// SIMATIC S7-200 project (STEP 7-Micro/WIN), CPU 224 REL 02.01

SYMBOL_TABLE USER1
oneLevel         VW2
twoLevel         VW3
onePres4ma       VW4
onePres20ma      VW5
twoPres4ma       VW6
twoPres20ma      VW7
oneUpp           VW8
oneLww           VW9
twoUpp           VW10
twoLww           VW11
pmp1mode         VW12     // 0 - stop, 1 - auto, 3 - man
pmp2mode         VW13
dOneLevel        VD14
dTwoLevel        VD16
dOnePres4ma      VD18
dOnePres20ma     VD20
dTwoPres4ma      VD22
dTwoPres20ma     VD24
dOneUpp          VD26
dOneLww          VD28
dTwoUpp          VD30
dTwoLww          VD32
pmp1auto         I0.0
pmp2auto         I0.1
pmp1man          I0.2
pmp2man          I0.3
pmp1turn         Q0.0
pmp2turn         Q0.1
oneMustStart     V34.0
twoMustStart     V34.1
pmp1state        V34.2
pmp2state        V34.3
END_SYMBOL_TABLE

ORGANIZATION_BLOCK MAIN:OB1
TITLE=PROGRAM COMMENTS
BEGIN
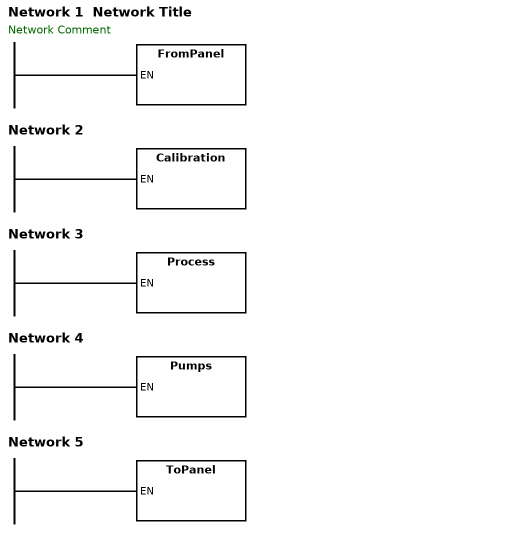
Network 1 // Network Title
// Network Comment
// (network saved uncompiled; LAD cells follow)
// row 0: c0 --  c1 [FromPanel EN:=power@row0]
Network 2
// (network saved uncompiled; LAD cells follow)
// row 0: c0 --  c1 [Calibration EN:=power@row0]
Network 3
// (network saved uncompiled; LAD cells follow)
// row 0: c0 --  c1 [Process EN:=power@row0]
Network 4
// (network saved uncompiled; LAD cells follow)
// row 0: c0 --  c1 [Pumps EN:=power@row0]
Network 5
// (network saved uncompiled; LAD cells follow)
// row 0: c0 --  c1 [ToPanel EN:=power@row0]
END_ORGANIZATION_BLOCK

SUBROUTINE_BLOCK Calibration:SBR0
TITLE=SUBROUTINE COMMENTS
BEGIN
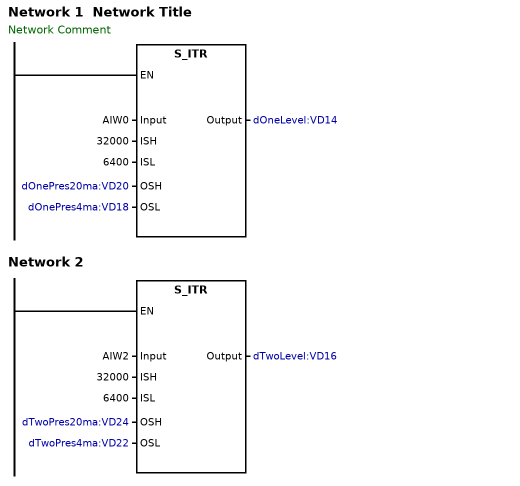
Network 1 // Network Title
// Network Comment
// (network saved uncompiled; LAD cells follow)
// row 0: c0 --  c1 [S_ITR EN:=power@row0, Input:=AIW0, ISH:=32000, ISL:=6400, OSH:=dOnePres20ma:VD20, OSL:=dOnePres4ma:VD18, Output=>dOneLevel:VD14]
// row 1: c1 [box]
// row 2: c1 [box]
Network 2
// (network saved uncompiled; LAD cells follow)
// row 0: c0 --  c1 [S_ITR EN:=power@row0, Input:=AIW2, ISH:=32000, ISL:=6400, OSH:=dTwoPres20ma:VD24, OSL:=dTwoPres4ma:VD22, Output=>dTwoLevel:VD16]
// row 1: c1 [box]
// row 2: c1 [box]
END_SUBROUTINE_BLOCK

SUBROUTINE_BLOCK FromPanel:SBR1
TITLE=SUBROUTINE COMMENTS
BEGIN
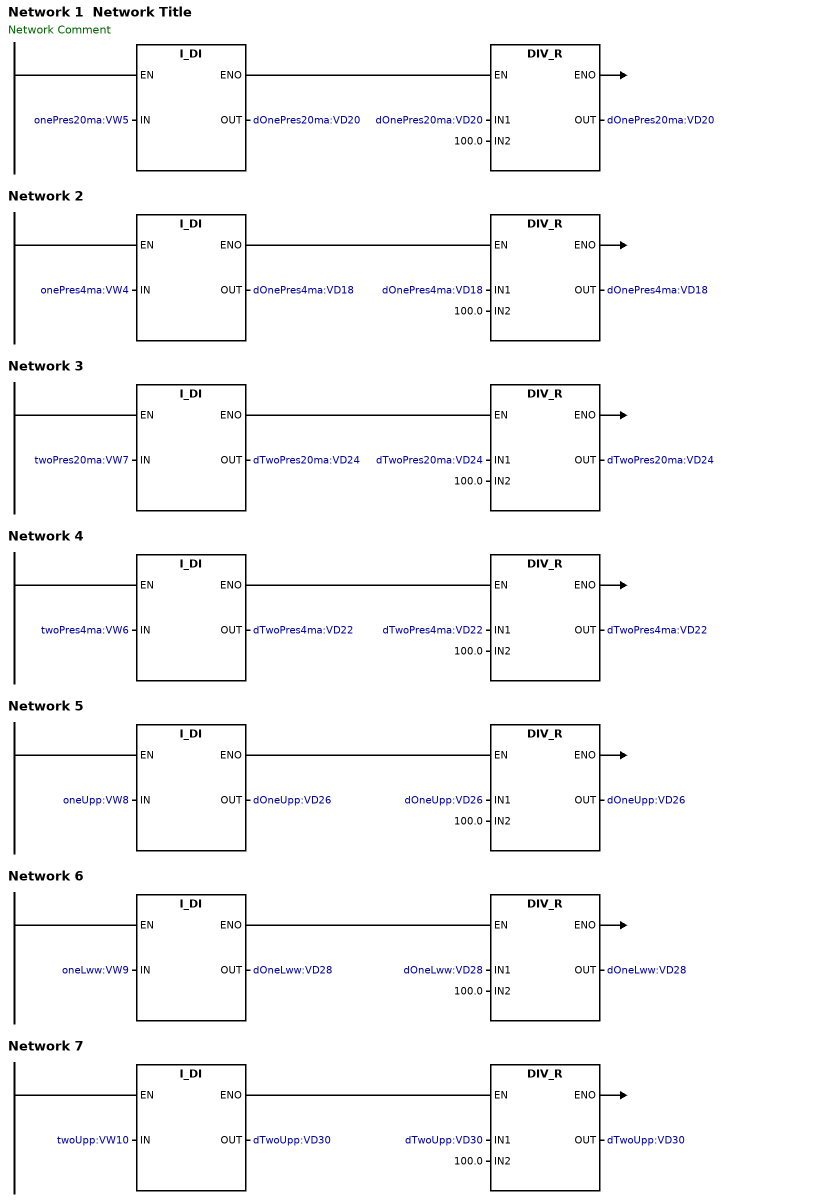
Network 1 // Network Title
// Network Comment
// (network saved uncompiled; LAD cells follow)
// row 0: c0 --  c1 [I_DI EN:=power@row0, IN:=onePres20ma:VW5, ENO=>power, OUT=>dOnePres20ma:VD20]  c2 --  c3 --  c4 [DIV_R EN:=power@row0, IN1:=dOnePres20ma:VD20, IN2:=100.0, ENO=>power, OUT=>dOnePres20ma:VD20]  c5 ->
// row 1: c1 [box]  c4 [box]
Network 2
// (network saved uncompiled; LAD cells follow)
// row 0: c0 --  c1 [I_DI EN:=power@row0, IN:=onePres4ma:VW4, ENO=>power, OUT=>dOnePres4ma:VD18]  c2 --  c3 --  c4 [DIV_R EN:=power@row0, IN1:=dOnePres4ma:VD18, IN2:=100.0, ENO=>power, OUT=>dOnePres4ma:VD18]  c5 ->
// row 1: c1 [box]  c4 [box]
Network 3
// (network saved uncompiled; LAD cells follow)
// row 0: c0 --  c1 [I_DI EN:=power@row0, IN:=twoPres20ma:VW7, ENO=>power, OUT=>dTwoPres20ma:VD24]  c2 --  c3 --  c4 [DIV_R EN:=power@row0, IN1:=dTwoPres20ma:VD24, IN2:=100.0, ENO=>power, OUT=>dTwoPres20ma:VD24]  c5 ->
// row 1: c1 [box]  c4 [box]
Network 4
// (network saved uncompiled; LAD cells follow)
// row 0: c0 --  c1 [I_DI EN:=power@row0, IN:=twoPres4ma:VW6, ENO=>power, OUT=>dTwoPres4ma:VD22]  c2 --  c3 --  c4 [DIV_R EN:=power@row0, IN1:=dTwoPres4ma:VD22, IN2:=100.0, ENO=>power, OUT=>dTwoPres4ma:VD22]  c5 ->
// row 1: c1 [box]  c4 [box]
Network 5
// (network saved uncompiled; LAD cells follow)
// row 0: c0 --  c1 [I_DI EN:=power@row0, IN:=oneUpp:VW8, ENO=>power, OUT=>dOneUpp:VD26]  c2 --  c3 --  c4 [DIV_R EN:=power@row0, IN1:=dOneUpp:VD26, IN2:=100.0, ENO=>power, OUT=>dOneUpp:VD26]  c5 ->
// row 1: c1 [box]  c4 [box]
Network 6
// (network saved uncompiled; LAD cells follow)
// row 0: c0 --  c1 [I_DI EN:=power@row0, IN:=oneLww:VW9, ENO=>power, OUT=>dOneLww:VD28]  c2 --  c3 --  c4 [DIV_R EN:=power@row0, IN1:=dOneLww:VD28, IN2:=100.0, ENO=>power, OUT=>dOneLww:VD28]  c5 ->
// row 1: c1 [box]  c4 [box]
Network 7
// (network saved uncompiled; LAD cells follow)
// row 0: c0 --  c1 [I_DI EN:=power@row0, IN:=twoUpp:VW10, ENO=>power, OUT=>dTwoUpp:VD30]  c2 --  c3 --  c4 [DIV_R EN:=power@row0, IN1:=dTwoUpp:VD30, IN2:=100.0, ENO=>power, OUT=>dTwoUpp:VD30]  c5 ->
// row 1: c1 [box]  c4 [box]
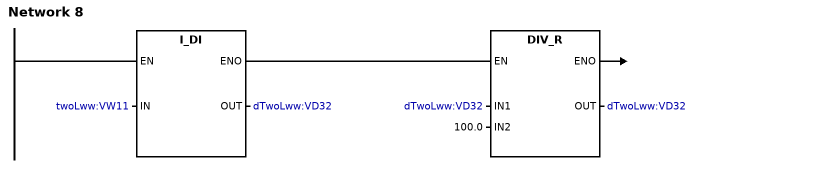
Network 8
// (network saved uncompiled; LAD cells follow)
// row 0: c0 --  c1 [I_DI EN:=power@row0, IN:=twoLww:VW11, ENO=>power, OUT=>dTwoLww:VD32]  c2 --  c3 --  c4 [DIV_R EN:=power@row0, IN1:=dTwoLww:VD32, IN2:=100.0, ENO=>power, OUT=>dTwoLww:VD32]  c5 ->
// row 1: c1 [box]  c4 [box]
END_SUBROUTINE_BLOCK

// SBR2: protected block, not included

SUBROUTINE_BLOCK Process:SBR3
TITLE=SUBROUTINE COMMENTS
BEGIN
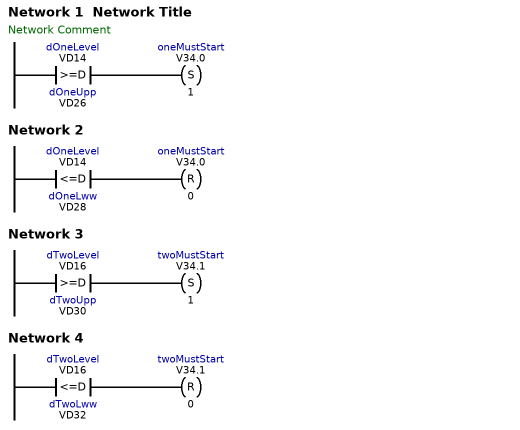
Network 1 // Network Title
// Network Comment
// (network saved uncompiled; LAD cells follow)
// row 0: c0 -|>=D|- dOneLevel:VD14, dOneUpp:VD26  c1 -(S) oneMustStart:V34.0, 1
Network 2
// (network saved uncompiled; LAD cells follow)
// row 0: c0 -|<=D|- dOneLevel:VD14, dOneLww:VD28  c1 -(R) oneMustStart:V34.0, 0
Network 3
// (network saved uncompiled; LAD cells follow)
// row 0: c0 -|>=D|- dTwoLevel:VD16, dTwoUpp:VD30  c1 -(S) twoMustStart:V34.1, 1
Network 4
// (network saved uncompiled; LAD cells follow)
// row 0: c0 -|<=D|- dTwoLevel:VD16, dTwoLww:VD32  c1 -(R) twoMustStart:V34.1, 0
END_SUBROUTINE_BLOCK

SUBROUTINE_BLOCK Pumps:SBR4
TITLE=SUBROUTINE COMMENTS
BEGIN
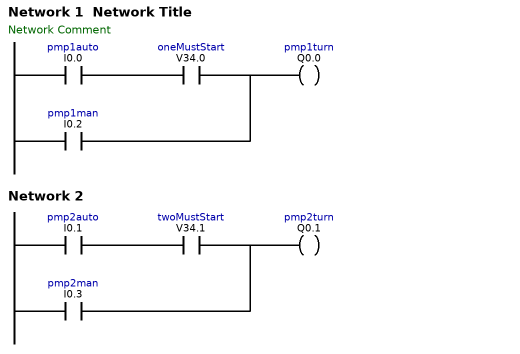
Network 1 // Network Title
// Network Comment
// (network saved uncompiled; LAD cells follow)
// row 0: c0 -| |- pmp1auto:I0.0  c1 -| |- oneMustStart:V34.0 v  c2 -( ) pmp1turn:Q0.0
// row 1: c0 -| |- pmp1man:I0.2  c1 -- ^
Network 2
// (network saved uncompiled; LAD cells follow)
// row 0: c0 -| |- pmp2auto:I0.1  c1 -| |- twoMustStart:V34.1 v  c2 -( ) pmp2turn:Q0.1
// row 1: c0 -| |- pmp2man:I0.3  c1 -- ^
END_SUBROUTINE_BLOCK

SUBROUTINE_BLOCK ToPanel:SBR5
TITLE=SUBROUTINE COMMENTS
BEGIN
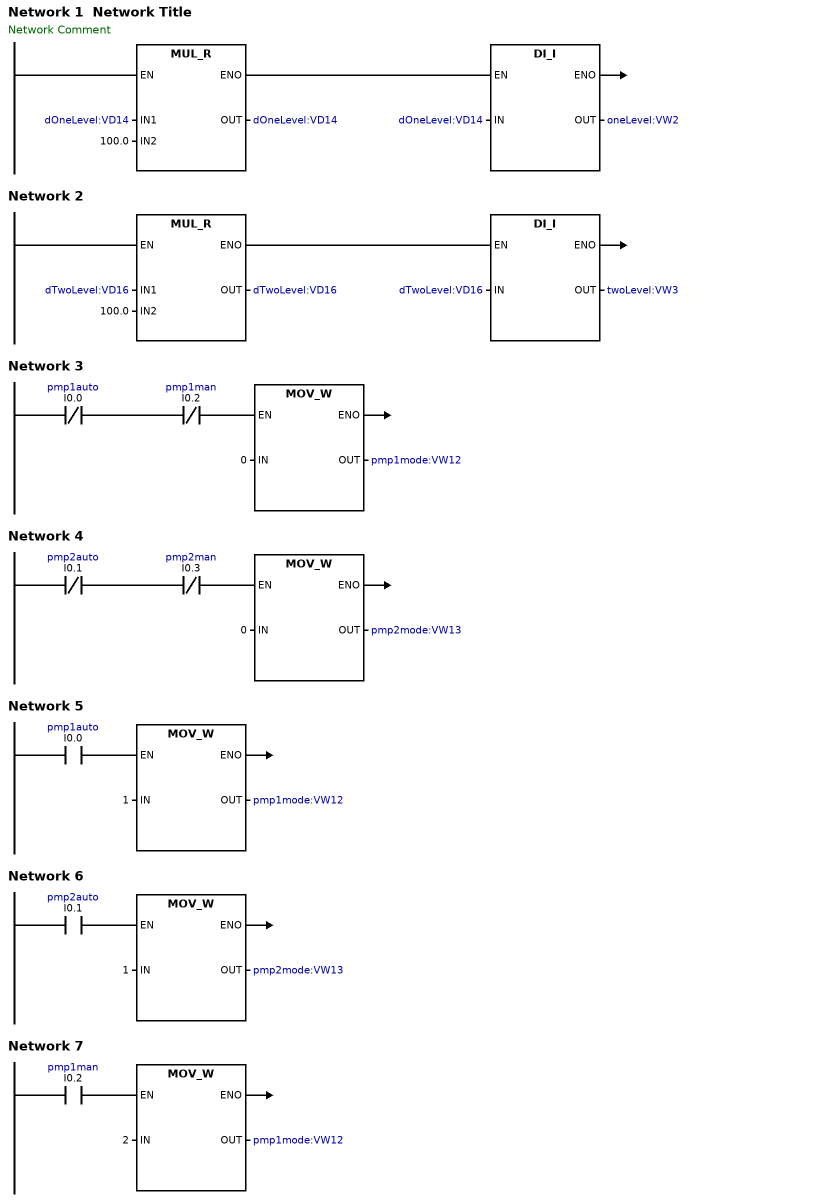
Network 1 // Network Title
// Network Comment
// (network saved uncompiled; LAD cells follow)
// row 0: c0 --  c1 [MUL_R EN:=power@row0, IN1:=dOneLevel:VD14, IN2:=100.0, ENO=>power, OUT=>dOneLevel:VD14]  c2 --  c3 --  c4 [DI_I EN:=power@row0, IN:=dOneLevel:VD14, ENO=>power, OUT=>oneLevel:VW2]  c5 ->
// row 1: c1 [box]  c4 [box]
Network 2
// (network saved uncompiled; LAD cells follow)
// row 0: c0 --  c1 [MUL_R EN:=power@row0, IN1:=dTwoLevel:VD16, IN2:=100.0, ENO=>power, OUT=>dTwoLevel:VD16]  c2 --  c3 --  c4 [DI_I EN:=power@row0, IN:=dTwoLevel:VD16, ENO=>power, OUT=>twoLevel:VW3]  c5 ->
// row 1: c1 [box]  c4 [box]
Network 3
// (network saved uncompiled; LAD cells follow)
// row 0: c0 -|/|- pmp1auto:I0.0  c1 -|/|- pmp1man:I0.2  c2 [MOV_W EN:=power@row0, IN:=0, ENO=>power, OUT=>pmp1mode:VW12]  c3 ->
// row 1: c2 [box]
Network 4
// (network saved uncompiled; LAD cells follow)
// row 0: c0 -|/|- pmp2auto:I0.1  c1 -|/|- pmp2man:I0.3  c2 [MOV_W EN:=power@row0, IN:=0, ENO=>power, OUT=>pmp2mode:VW13]  c3 ->
// row 1: c2 [box]
Network 5
// (network saved uncompiled; LAD cells follow)
// row 0: c0 -| |- pmp1auto:I0.0  c1 [MOV_W EN:=power@row0, IN:=1, ENO=>power, OUT=>pmp1mode:VW12]  c2 ->
// row 1: c1 [box]
Network 6
// (network saved uncompiled; LAD cells follow)
// row 0: c0 -| |- pmp2auto:I0.1  c1 [MOV_W EN:=power@row0, IN:=1, ENO=>power, OUT=>pmp2mode:VW13]  c2 ->
// row 1: c1 [box]
Network 7
// (network saved uncompiled; LAD cells follow)
// row 0: c0 -| |- pmp1man:I0.2  c1 [MOV_W EN:=power@row0, IN:=2, ENO=>power, OUT=>pmp1mode:VW12]  c2 ->
// row 1: c1 [box]
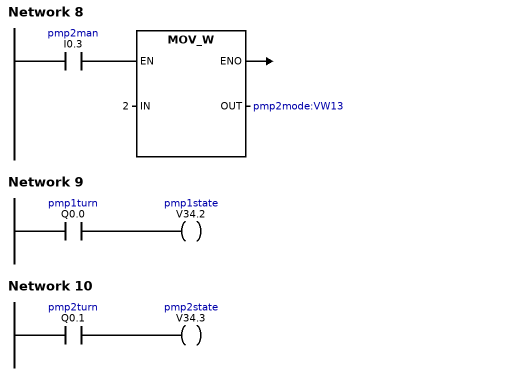
Network 8
// (network saved uncompiled; LAD cells follow)
// row 0: c0 -| |- pmp2man:I0.3  c1 [MOV_W EN:=power@row0, IN:=2, ENO=>power, OUT=>pmp2mode:VW13]  c2 ->
// row 1: c1 [box]
Network 9
// (network saved uncompiled; LAD cells follow)
// row 0: c0 -| |- pmp1turn:Q0.0  c1 -( ) pmp1state:V34.2
Network 10
// (network saved uncompiled; LAD cells follow)
// row 0: c0 -| |- pmp2turn:Q0.1  c1 -( ) pmp2state:V34.3
END_SUBROUTINE_BLOCK
